PROGRAM SafetyInterface_Enc062
VAR
	{attribute 'TcLinkTo' := '
		.iSafteyCtrlProjectCRC := TIIB[N70S14 (EL6910)]^Device Info Data^Project CRC;
		.iSafetyGroup_State := TIIB[N70S14 (EL6910)]^TwinSAFE Group Info Data^Enc062_SafetyGroup Info Data^State;
		.iSafetyGroup_Diag := TIIB[N70S14 (EL6910)]^TwinSAFE Group Info Data^Enc062_SafetyGroup Info Data^Diag;
		.iSafetyGroup_ComErr := TIIB[N70S14 (EL6910)]^StandardInputs^Enc062_SafetyGroup.oGroup_ComErr_3;
		.iSafetyGroup_ComInStartup := TIIB[N70S14 (EL6910)]^StandardInputs^Enc062_SafetyGroup.oGroup_ComInStartup_4;
		.iSafetyGroup_FBErr := TIIB[N70S14 (EL6910)]^StandardInputs^Enc062_SafetyGroup.oGroup_FBErr_5;
		.iSafetyGroup_FBInRun := TIIB[N70S14 (EL6910)]^StandardInputs^Enc062_SafetyGroup.oGroup_FBInRun_6;
		.iSafetyGroup_InRun := TIIB[N70S14 (EL6910)]^StandardInputs^Enc062_SafetyGroup.oGroup_InRun_7;
		.iSafetyGroup_OtherErr := TIIB[N70S14 (EL6910)]^StandardInputs^Enc062_SafetyGroup.oGroup_OtherErr_8;
		.oSafetyGroup_ErrAck := TIIB[N70S14 (EL6910)]^StandardOutputs^Enc062_SafetyGroup.iGroup_ErrAck_1;
		.oSafetyGroup_Run := TIIB[N70S14 (EL6910)]^StandardOutputs^Enc062_SafetyGroup.iGroup_Run_2;
		.oControlPowerPBLight := TIIB[N70S09 (EL2008)]^Channel 1^Output;
		.iSafetyResetPB := TIIB[N70S14 (EL6910)]^Connection Info Data^Enc062_SafetyGroup.N70S01 Digital 4 In (EL1904)_9 Info Data^Input Safe Data InputChannel3;
		.iEstopPB1_CH1 := TIIB[N70S14 (EL6910)]^Connection Info Data^Enc062_SafetyGroup.N70S01 Digital 4 In (EL1904)_9 Info Data^Input Safe Data InputChannel1;
		.iEstopPB1_CH2 := TIIB[N70S14 (EL6910)]^Connection Info Data^Enc062_SafetyGroup.N70S01 Digital 4 In (EL1904)_9 Info Data^Input Safe Data InputChannel2;
		.iRelayNCContact_Estop := TIIB[N70S14 (EL6910)]^Connection Info Data^Enc062_SafetyGroup.N70S03 Digital 4 In (EL1904)_11 Info Data^Input Safe Data InputChannel1;
		.iSafetyPowerOn_Estop_CH1 := TIIB[N70S14 (EL6910)]^Connection Info Data^Enc062_SafetyGroup.N70S04 Digital 4 Out (EL2904)_20 Info Data^Output Safe Data OutputChannel1;
		.iSafetyPowerOn_Estop_CH2 := TIIB[N70S14 (EL6910)]^Connection Info Data^Enc062_SafetyGroup.N70S04 Digital 4 Out (EL2904)_20 Info Data^Output Safe Data OutputChannel2;
		.iAirPressureOk := TIIB[N70S06 (EL1008)]^Channel 2^Input'}
	fbSafetyInterface : FB_SafetyInterfaceConv;
END_VAR



fbSafetyInterface(
	pSafetyInterface := ADR(gProduced_SafetyInterfaceConv.Enc062));

END_PROGRAM

(* stored: Version 1.1.0.1, ProductVersion 3.1.4024.6
   POU SafetyInterface_Enc062: Id {9469d990-49b8-4e3e-9f72-fd346f6cd078}, SpecialFunc None *)
